# EPICS substitutions: epicsApp/db/CAENHV2-14.substitutions
file "db/CAENHV_A.template" {
   {crate=2, slot=14, BoardType=SY1527, IP=192.168.30.11, ChMax=24}
}
file "db/CAENHV_B.template" {
   { crate=2, slot=14, name=BdStatus,    ch=1   }
   { crate=2, slot=14, name=CH0:V0Set,   ch=2   }
   { crate=2, slot=14, name=CH0:I0Set,   ch=3   }
   { crate=2, slot=14, name=CH0:VMon,    ch=4   }
   { crate=2, slot=14, name=CH0:IMon,    ch=5   }
   { crate=2, slot=14, name=CH0:Pw,      ch=6   }
   { crate=2, slot=14, name=CH0:Status,  ch=7   }
   { crate=2, slot=14, name=CH1:V0Set,   ch=8   }
   { crate=2, slot=14, name=CH1:I0Set,   ch=9   }
   { crate=2, slot=14, name=CH1:VMon,    ch=10  }
   { crate=2, slot=14, name=CH1:IMon,    ch=11  }
   { crate=2, slot=14, name=CH1:Pw,      ch=12  }
   { crate=2, slot=14, name=CH1:Status,  ch=13  }
   { crate=2, slot=14, name=CH2:V0Set,   ch=14  }
   { crate=2, slot=14, name=CH2:I0Set,   ch=15  }
   { crate=2, slot=14, name=CH2:VMon,    ch=16  }
   { crate=2, slot=14, name=CH2:IMon,    ch=17  }
   { crate=2, slot=14, name=CH2:Pw,      ch=18  }
   { crate=2, slot=14, name=CH2:Status,  ch=19  }
   { crate=2, slot=14, name=CH3:V0Set,   ch=20  }
   { crate=2, slot=14, name=CH3:I0Set,   ch=21  }
   { crate=2, slot=14, name=CH3:VMon,    ch=22  }
   { crate=2, slot=14, name=CH3:IMon,    ch=23  }
   { crate=2, slot=14, name=CH3:Pw,      ch=24  }
   { crate=2, slot=14, name=CH3:Status,  ch=25  }
   { crate=2, slot=14, name=CH4:V0Set,   ch=26  }
   { crate=2, slot=14, name=CH4:I0Set,   ch=27  }
   { crate=2, slot=14, name=CH4:VMon,    ch=28  }
   { crate=2, slot=14, name=CH4:IMon,    ch=29  }
   { crate=2, slot=14, name=CH4:Pw,      ch=30  }
   { crate=2, slot=14, name=CH4:Status,  ch=31  }
   { crate=2, slot=14, name=CH5:V0Set,   ch=32  }
   { crate=2, slot=14, name=CH5:I0Set,   ch=33  }
   { crate=2, slot=14, name=CH5:VMon,    ch=34  }
   { crate=2, slot=14, name=CH5:IMon,    ch=35  }
   { crate=2, slot=14, name=CH5:Pw,      ch=36  }
   { crate=2, slot=14, name=CH5:Status,  ch=37  }
   { crate=2, slot=14, name=CH6:V0Set,   ch=38  }
   { crate=2, slot=14, name=CH6:I0Set,   ch=39  }
   { crate=2, slot=14, name=CH6:VMon,    ch=40  }
   { crate=2, slot=14, name=CH6:IMon,    ch=41  }
   { crate=2, slot=14, name=CH6:Pw,      ch=42  }
   { crate=2, slot=14, name=CH6:Status,  ch=43  }
   { crate=2, slot=14, name=CH7:V0Set,   ch=44  }
   { crate=2, slot=14, name=CH7:I0Set,   ch=45  }
   { crate=2, slot=14, name=CH7:VMon,    ch=46  }
   { crate=2, slot=14, name=CH7:IMon,    ch=47  }
   { crate=2, slot=14, name=CH7:Pw,      ch=48  }
   { crate=2, slot=14, name=CH7:Status,  ch=49  }
   { crate=2, slot=14, name=CH8:V0Set,   ch=50  }
   { crate=2, slot=14, name=CH8:I0Set,   ch=51  }
   { crate=2, slot=14, name=CH8:VMon,    ch=52  }
   { crate=2, slot=14, name=CH8:IMon,    ch=53  }
   { crate=2, slot=14, name=CH8:Pw,      ch=54  }
   { crate=2, slot=14, name=CH8:Status,  ch=55  }
   { crate=2, slot=14, name=CH9:V0Set,   ch=56  }
   { crate=2, slot=14, name=CH9:I0Set,   ch=57  }
   { crate=2, slot=14, name=CH9:VMon,    ch=58  }
   { crate=2, slot=14, name=CH9:IMon,    ch=59  }
   { crate=2, slot=14, name=CH9:Pw,      ch=60  }
   { crate=2, slot=14, name=CH9:Status,  ch=61  }
   { crate=2, slot=14, name=CH10:V0Set,  ch=62  }
   { crate=2, slot=14, name=CH10:I0Set,  ch=63  }
   { crate=2, slot=14, name=CH10:VMon,   ch=64  }
   { crate=2, slot=14, name=CH10:IMon,   ch=65  }
   { crate=2, slot=14, name=CH10:Pw,     ch=66  }
   { crate=2, slot=14, name=CH10:Status, ch=67  }
   { crate=2, slot=14, name=CH11:V0Set,  ch=68  }
   { crate=2, slot=14, name=CH11:I0Set,  ch=69  }
   { crate=2, slot=14, name=CH11:VMon,   ch=70  }
   { crate=2, slot=14, name=CH11:IMon,   ch=71  }
   { crate=2, slot=14, name=CH11:Pw,     ch=72  }
   { crate=2, slot=14, name=CH11:Status, ch=73  }
   { crate=2, slot=14, name=CH12:V0Set,  ch=74  }
   { crate=2, slot=14, name=CH12:I0Set,  ch=75  }
   { crate=2, slot=14, name=CH12:VMon,   ch=76  }
   { crate=2, slot=14, name=CH12:IMon,   ch=77  }
   { crate=2, slot=14, name=CH12:Pw,     ch=78  }
   { crate=2, slot=14, name=CH12:Status, ch=79  }
   { crate=2, slot=14, name=CH13:V0Set,  ch=80  }
   { crate=2, slot=14, name=CH13:I0Set,  ch=81  }
   { crate=2, slot=14, name=CH13:VMon,   ch=82  }
   { crate=2, slot=14, name=CH13:IMon,   ch=83  }
   { crate=2, slot=14, name=CH13:Pw,     ch=84  }
   { crate=2, slot=14, name=CH13:Status, ch=85  }
   { crate=2, slot=14, name=CH14:V0Set,  ch=86  }
   { crate=2, slot=14, name=CH14:I0Set,  ch=87  }
   { crate=2, slot=14, name=CH14:VMon,   ch=88  }
   { crate=2, slot=14, name=CH14:IMon,   ch=89  }
   { crate=2, slot=14, name=CH14:Pw,     ch=90  }
   { crate=2, slot=14, name=CH14:Status, ch=91  }
   { crate=2, slot=14, name=CH15:V0Set,  ch=92  }
   { crate=2, slot=14, name=CH15:I0Set,  ch=93  }
   { crate=2, slot=14, name=CH15:VMon,   ch=94  }
   { crate=2, slot=14, name=CH15:IMon,   ch=95  }
   { crate=2, slot=14, name=CH15:Pw,     ch=96  }
   { crate=2, slot=14, name=CH15:Status, ch=97  }
   { crate=2, slot=14, name=CH16:V0Set,  ch=98  }
   { crate=2, slot=14, name=CH16:I0Set,  ch=99  }
   { crate=2, slot=14, name=CH16:VMon,   ch=100 }
   { crate=2, slot=14, name=CH16:IMon,   ch=101 }
   { crate=2, slot=14, name=CH16:Pw,     ch=102 }
   { crate=2, slot=14, name=CH16:Status, ch=103 }
   { crate=2, slot=14, name=CH17:V0Set,  ch=104 }
   { crate=2, slot=14, name=CH17:I0Set,  ch=105 }
   { crate=2, slot=14, name=CH17:VMon,   ch=106 }
   { crate=2, slot=14, name=CH17:IMon,   ch=107 }
   { crate=2, slot=14, name=CH17:Pw,     ch=108 }
   { crate=2, slot=14, name=CH17:Status, ch=109 }
   { crate=2, slot=14, name=CH18:V0Set,  ch=110 }
   { crate=2, slot=14, name=CH18:I0Set,  ch=111 }
   { crate=2, slot=14, name=CH18:VMon,   ch=112 }
   { crate=2, slot=14, name=CH18:IMon,   ch=113 }
   { crate=2, slot=14, name=CH18:Pw,     ch=114 }
   { crate=2, slot=14, name=CH18:Status, ch=115 }
   { crate=2, slot=14, name=CH19:V0Set,  ch=116 }
   { crate=2, slot=14, name=CH19:I0Set,  ch=117 }
   { crate=2, slot=14, name=CH19:VMon,   ch=118 }
   { crate=2, slot=14, name=CH19:IMon,   ch=119 }
   { crate=2, slot=14, name=CH19:Pw,     ch=120 }
   { crate=2, slot=14, name=CH19:Status, ch=121 }
   { crate=2, slot=14, name=CH20:V0Set,  ch=122 }
   { crate=2, slot=14, name=CH20:I0Set,  ch=123 }
   { crate=2, slot=14, name=CH20:VMon,   ch=124 }
   { crate=2, slot=14, name=CH20:IMon,   ch=125 }
   { crate=2, slot=14, name=CH20:Pw,     ch=126 }
   { crate=2, slot=14, name=CH20:Status, ch=127 }
   { crate=2, slot=14, name=CH21:V0Set,  ch=128 }
   { crate=2, slot=14, name=CH21:I0Set,  ch=129 }
   { crate=2, slot=14, name=CH21:VMon,   ch=130 }
   { crate=2, slot=14, name=CH21:IMon,   ch=131 }
   { crate=2, slot=14, name=CH21:Pw,     ch=132 }
   { crate=2, slot=14, name=CH21:Status, ch=133 }
   { crate=2, slot=14, name=CH22:V0Set,  ch=134 }
   { crate=2, slot=14, name=CH22:I0Set,  ch=135 }
   { crate=2, slot=14, name=CH22:VMon,   ch=136 }
   { crate=2, slot=14, name=CH22:IMon,   ch=137 }
   { crate=2, slot=14, name=CH22:Pw,     ch=138 }
   { crate=2, slot=14, name=CH22:Status, ch=139 }
   { crate=2, slot=14, name=CH23:V0Set,  ch=140 }
   { crate=2, slot=14, name=CH23:I0Set,  ch=141 }
   { crate=2, slot=14, name=CH23:VMon,   ch=142 }
   { crate=2, slot=14, name=CH23:IMon,   ch=143 }
   { crate=2, slot=14, name=CH23:Pw,     ch=144 }
   { crate=2, slot=14, name=CH23:Status, ch=145 }
}
